PROGRAM POUfbd
VAR_INPUT
    mxManRunOk : BOOL;
    mxAutoRunOk : BOOL;
    ixBtnAout : BOOL;
    ixBtnAin  : BOOL;
    ixBtnBout : BOOL;
    ixBtnBin  : BOOL;
    ixBtnDrillOut : BOOL;
    ixBtnDrillIn  : BOOL;
END_VAR
VAR_INPUT
    mxAutoAout      : BOOL;
    mxAutoAin       : BOOL;
    mxAutoBout      : BOOL;
    mxAutoBin       : BOOL;
    mxAutoDrillDown : BOOL;
    mxAutoDrillUp   : BOOL;
END_VAR
VAR_OUTPUT
    qxSliderAout : BOOL;
    qxSliderAin  : BOOL;
    qxSliderBout : BOOL;
    qxSliderBin  : BOOL;
    qxDrillDown  : BOOL;
    qxDrillUp    : BOOL;
END_VAR
VAR
	fbBlink : BLINK;
    mxBlink : BOOL;
	mxSumSafetytopReady: BOOL;
	mxSafetyStopOk: BOOL;
	qxLampEmStopOk: BOOL;
	mxEmStopOk: BOOL;
	ixBtnReset: BOOL;
	ixSafety1StopOk: BOOL;
	ixSafety2StopOk: BOOL;
	ixAuto: BOOL;	
	mxAutoModeReady: BOOL;
	ixSliderAin: BOOL;
	ixSlideBout: BOOL;
	ixDrillUp: BOOL;
	qxLampHomePos: BOOL;
	ixButtonStop: BOOL;
	mxCycleStopActivated: BOOL;
	ixButtonStart: BOOL;
	mxCycleStop: BOOL;
	qxLampStarted: BOOL;
	mxAutoDrillOut: BOOL;
END_VAR

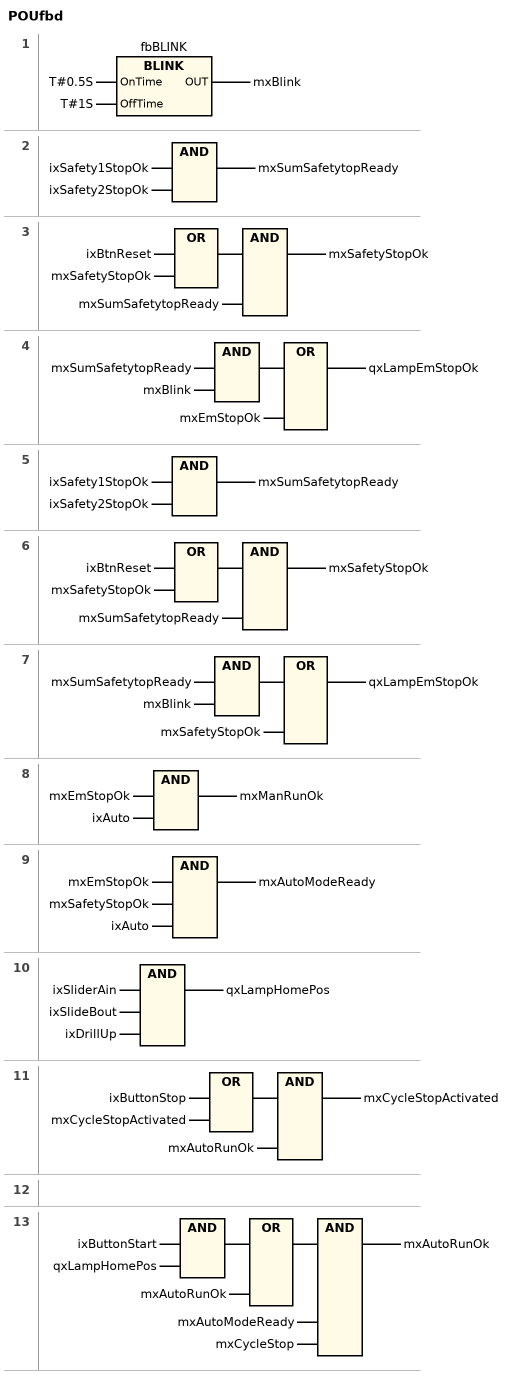
// NETWORK 1
fbBLINK(OnTime := T#0.5S, OffTime := T#1S); // BLINK
mxBlink := fbBLINK.OUT;

// NETWORK 2
mxSumSafetytopReady := ixSafety1StopOk AND ixSafety2StopOk;

// NETWORK 3
mxSafetyStopOk := (ixBtnReset OR mxSafetyStopOk) AND mxSumSafetytopReady;

// NETWORK 4
qxLampEmStopOk := mxSumSafetytopReady AND mxBlink OR mxEmStopOk;

// NETWORK 5
mxSumSafetytopReady := ixSafety1StopOk AND ixSafety2StopOk;

// NETWORK 6
mxSafetyStopOk := (ixBtnReset OR mxSafetyStopOk) AND mxSumSafetytopReady;

// NETWORK 7
qxLampEmStopOk := mxSumSafetytopReady AND mxBlink OR mxSafetyStopOk;

// NETWORK 8
mxManRunOk := mxEmStopOk AND ixAuto;

// NETWORK 9
mxAutoModeReady := mxEmStopOk AND mxSafetyStopOk AND ixAuto;

// NETWORK 10
qxLampHomePos := ixSliderAin AND ixSlideBout AND ixDrillUp;

// NETWORK 11
mxCycleStopActivated := (ixButtonStop OR mxCycleStopActivated) AND mxAutoRunOk;

// NETWORK 12

// NETWORK 13
mxAutoRunOk := (ixButtonStart AND qxLampHomePos OR mxAutoRunOk) AND mxAutoModeReady AND mxCycleStop;

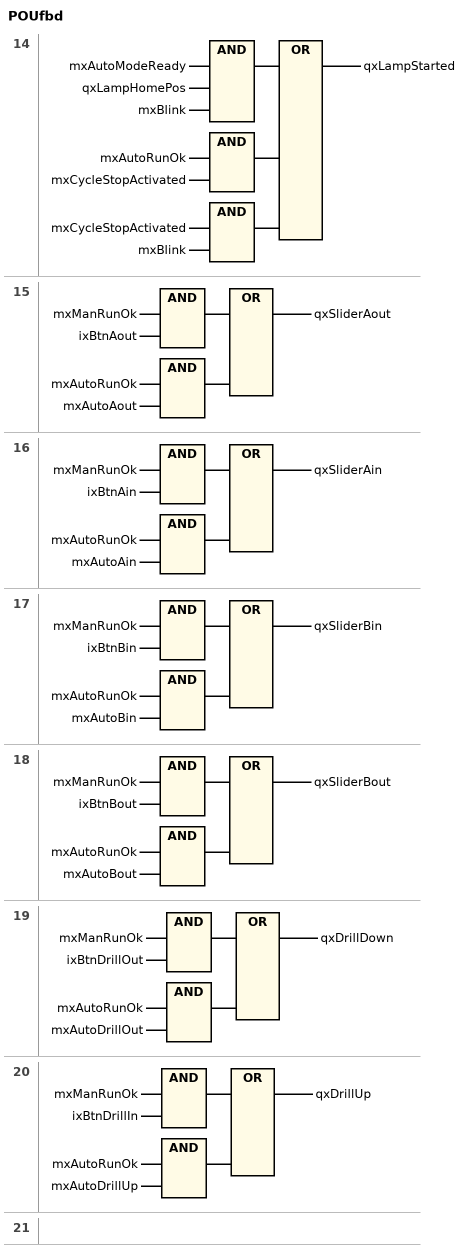
// NETWORK 14
qxLampStarted := mxAutoModeReady AND qxLampHomePos AND mxBlink OR mxAutoRunOk AND mxCycleStopActivated OR mxCycleStopActivated AND mxBlink;

// NETWORK 15
qxSliderAout := mxManRunOk AND ixBtnAout OR mxAutoRunOk AND mxAutoAout;

// NETWORK 16
qxSliderAin := mxManRunOk AND ixBtnAin OR mxAutoRunOk AND mxAutoAin;

// NETWORK 17
qxSliderBin := mxManRunOk AND ixBtnBin OR mxAutoRunOk AND mxAutoBin;

// NETWORK 18
qxSliderBout := mxManRunOk AND ixBtnBout OR mxAutoRunOk AND mxAutoBout;

// NETWORK 19
qxDrillDown := mxManRunOk AND ixBtnDrillOut OR mxAutoRunOk AND mxAutoDrillOut;

// NETWORK 20
qxDrillUp := mxManRunOk AND ixBtnDrillIn OR mxAutoRunOk AND mxAutoDrillUp;

// NETWORK 21

END_PROGRAM

(* stored: Version 1.1.0.1
   POU POUfbd: Id {f35513ce-5fbe-4cbd-af6c-bdd5a9aa24f4}, SpecialFunc None *)
